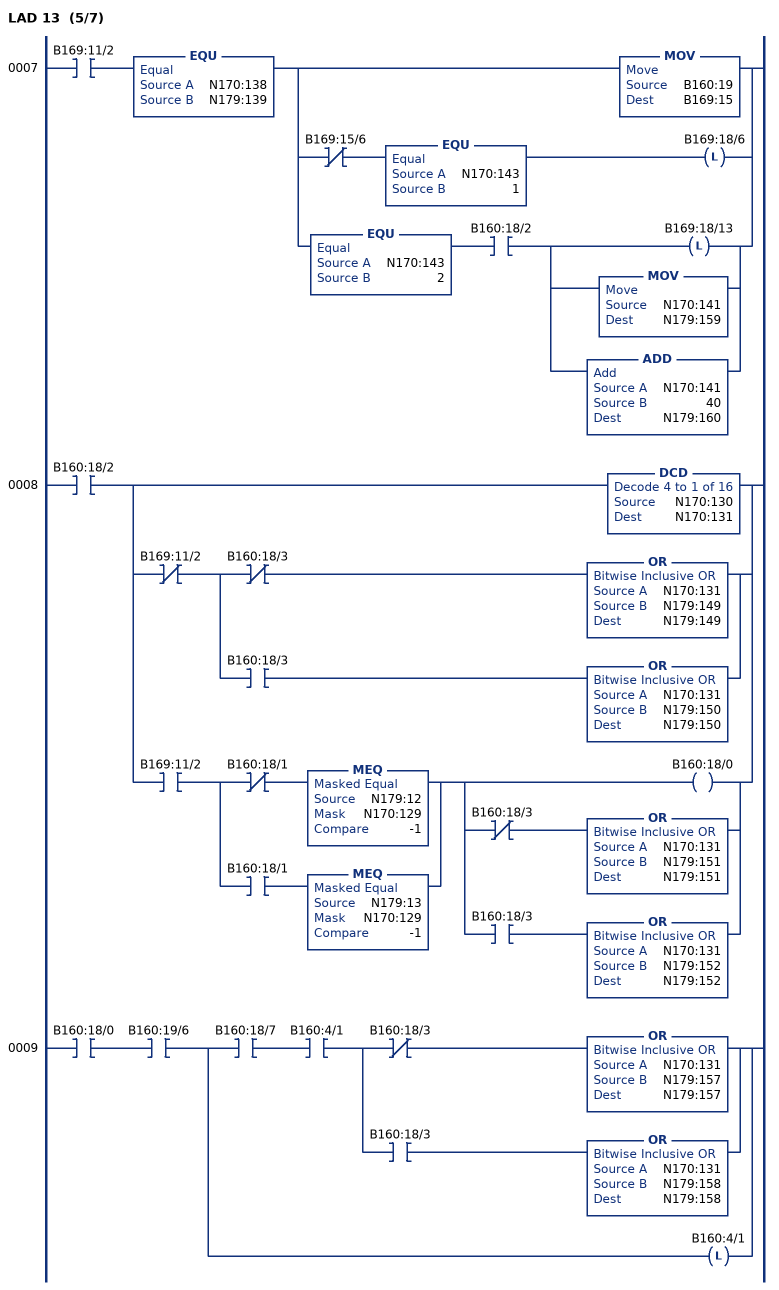
% Rung: 7 %
SOR XIC B169:11/2 EQU N170:138 N179:139 BST MOV B160:19 B169:15 NXB XIO B169:15/6 EQU N170:143 1 OTL B169:18/6 NXB EQU N170:143 2 XIC B160:18/2 BST OTL B169:18/13 NXB MOV N170:141 N179:159 NXB ADD N170:141 40 N179:160 BND BND EOR
% Rung: 8 %
SOR XIC B160:18/2 BST DCD N170:130 N170:131 NXB XIO B169:11/2 BST XIO B160:18/3 OR N170:131 N179:149 N179:149 NXB XIC B160:18/3 OR N170:131 N179:150 N179:150 BND NXB XIC B169:11/2 BST XIO B160:18/1 MEQ N179:12 N170:129 -1 NXB XIC B160:18/1 MEQ N179:13 N170:129 -1 BND BST OTE B160:18/0 NXB XIO B160:18/3 OR N170:131 N179:151 N179:151 NXB XIC B160:18/3 OR N170:131 N179:152 N179:152 BND BND EOR
% Rung: 9 %
SOR XIC B160:18/0 XIC B160:19/6 BST XIC B160:18/7 XIC B160:4/1 BST XIO B160:18/3 OR N170:131 N179:157 N179:157 NXB XIC B160:18/3 OR N170:131 N179:158 N179:158 BND NXB OTL B160:4/1 BND EOR

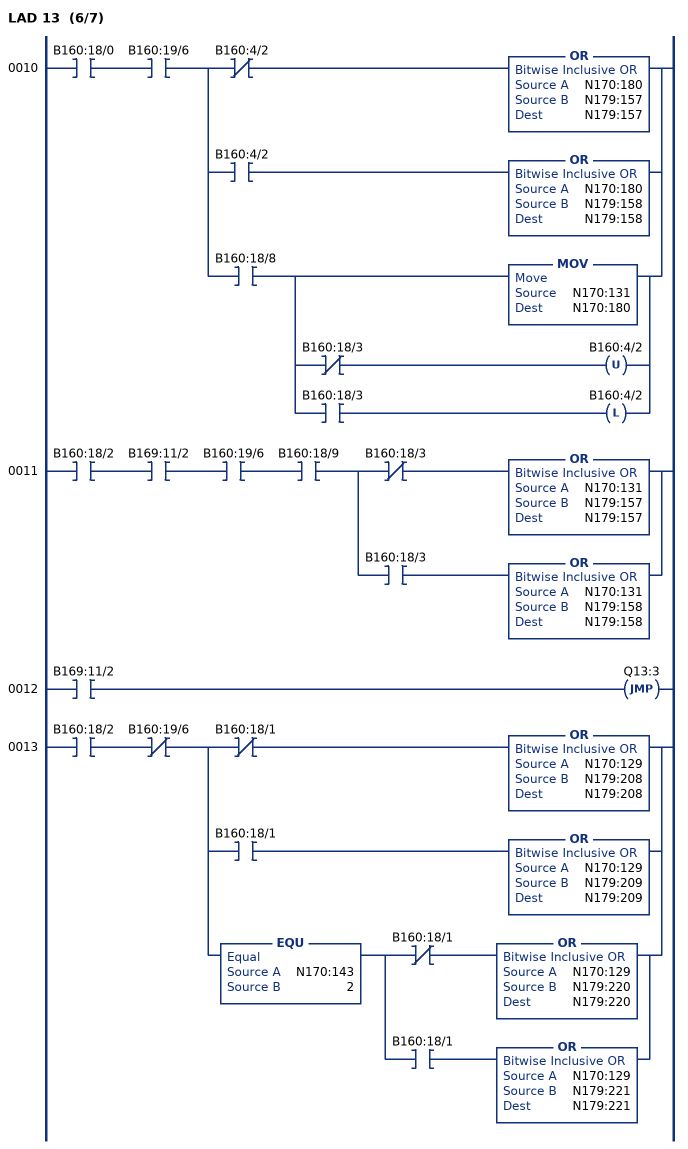
% Rung: 10 %
SOR XIC B160:18/0 XIC B160:19/6 BST BST XIO B160:4/2 OR N170:180 N179:157 N179:157 NXB XIC B160:4/2 OR N170:180 N179:158 N179:158 BND NXB XIC B160:18/8 BST MOV N170:131 N170:180 NXB XIO B160:18/3 OTU B160:4/2 NXB XIC B160:18/3 OTL B160:4/2 BND BND EOR
% Rung: 11 %
SOR XIC B160:18/2 XIC B169:11/2 XIC B160:19/6 XIC B160:18/9 BST XIO B160:18/3 OR N170:131 N179:157 N179:157 NXB XIC B160:18/3 OR N170:131 N179:158 N179:158 BND EOR
% Rung: 12 %
SOR XIC B169:11/2 JMP Q13:3 EOR
% Rung: 13 %
SOR XIC B160:18/2 XIO B160:19/6 BST BST XIO B160:18/1 OR N170:129 N179:208 N179:208 NXB XIC B160:18/1 OR N170:129 N179:209 N179:209 BND NXB EQU N170:143 2 BST XIO B160:18/1 OR N170:129 N179:220 N179:220 NXB XIC B160:18/1 OR N170:129 N179:221 N179:221 BND BND EOR

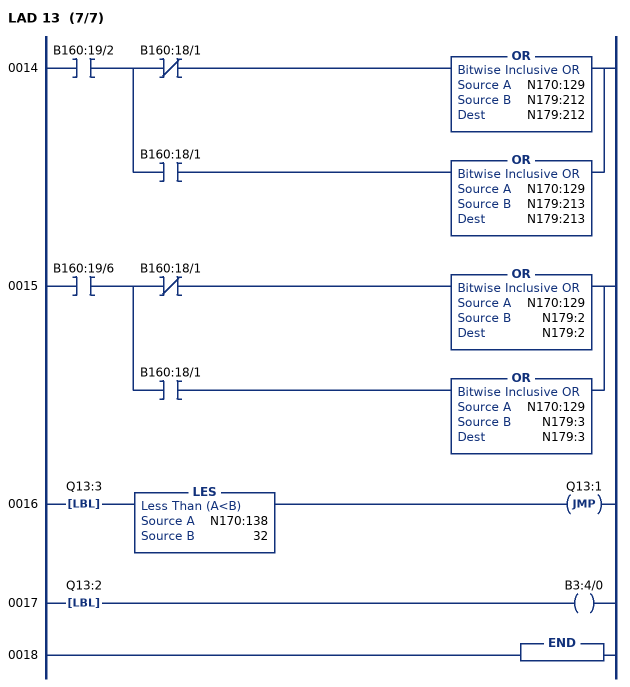
% Rung: 14 %
SOR XIC B160:19/2 BST XIO B160:18/1 OR N170:129 N179:212 N179:212 NXB XIC B160:18/1 OR N170:129 N179:213 N179:213 BND EOR
% Rung: 15 %
SOR XIC B160:19/6 BST XIO B160:18/1 OR N170:129 N179:2 N179:2 NXB XIC B160:18/1 OR N170:129 N179:3 N179:3 BND EOR
% Rung: 16 %
SOR LBL Q13:3 LES N170:138 32 JMP Q13:1 EOR
% Rung: 17 %
SOR LBL Q13:2 OTE B3:4/0 EOR
% Rung: 18 %
SOR END EOR

LADDER 15
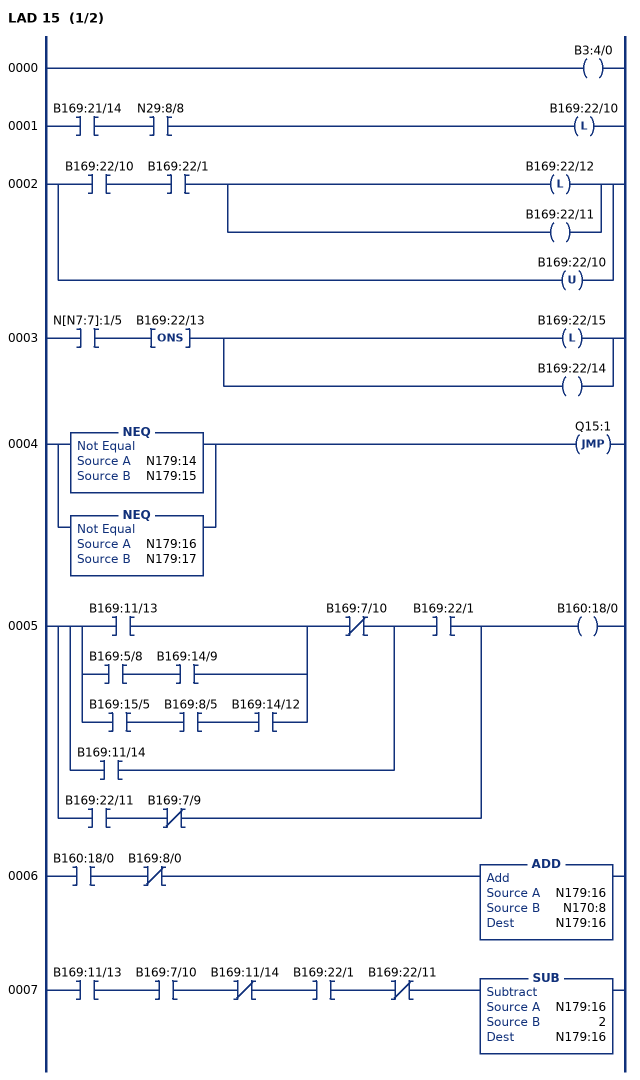
% Rung: 0 %
SOR OTE B3:4/0 EOR
% Rung: 1 %
SOR XIC B169:21/14 XIC N29:8/8 OTL B169:22/10 EOR
% Rung: 2 %
SOR BST XIC B169:22/10 XIC B169:22/1 BST OTL B169:22/12 NXB OTE B169:22/11 BND NXB OTU B169:22/10 BND EOR
% Rung: 3 %
SOR XIC N[N7:7]:1/5 OSR B169:22/13 BST OTL B169:22/15 NXB OTE B169:22/14 BND EOR
% Rung: 4 %
SOR BST NEQ N179:14 N179:15 NXB NEQ N179:16 N179:17 BND JMP Q15:1 EOR
% Rung: 5 %
SOR BST BST BST XIC B169:11/13 NXB XIC B169:5/8 XIC B169:14/9 NXB XIC B169:15/5 XIC B169:8/5 XIC B169:14/12 BND XIO B169:7/10 NXB XIC B169:11/14 BND XIC B169:22/1 NXB XIC B169:22/11 XIO B169:7/9 BND OTE B160:18/0 EOR
% Rung: 6 %
SOR XIC B160:18/0 XIO B169:8/0 ADD N179:16 N170:8 N179:16 EOR
% Rung: 7 %
SOR XIC B169:11/13 XIC B169:7/10 XIO B169:11/14 XIC B169:22/1 XIO B169:22/11 SUB N179:16 2 N179:16 EOR

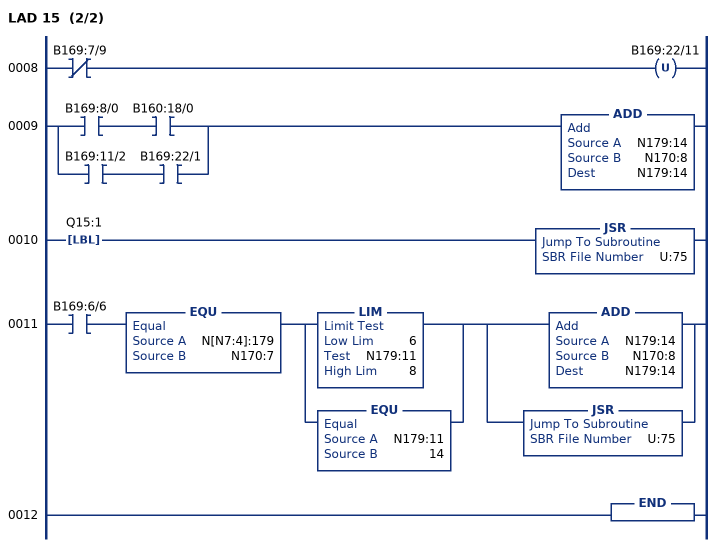
% Rung: 8 %
SOR XIO B169:7/9 OTU B169:22/11 EOR
% Rung: 9 %
SOR BST XIC B169:8/0 XIC B160:18/0 NXB XIC B169:11/2 XIC B169:22/1 BND ADD N179:14 N170:8 N179:14 EOR
% Rung: 10 %
SOR LBL Q15:1 JSR U:75 EOR
% Rung: 11 %
SOR XIC B169:6/6 EQU N[N7:4]:179 N170:7 BST LIM 6 N179:11 8 NXB EQU N179:11 14 BND BST ADD N179:14 N170:8 N179:14 NXB JSR U:75 BND EOR
% Rung: 12 %
SOR END EOR

LADDER 16
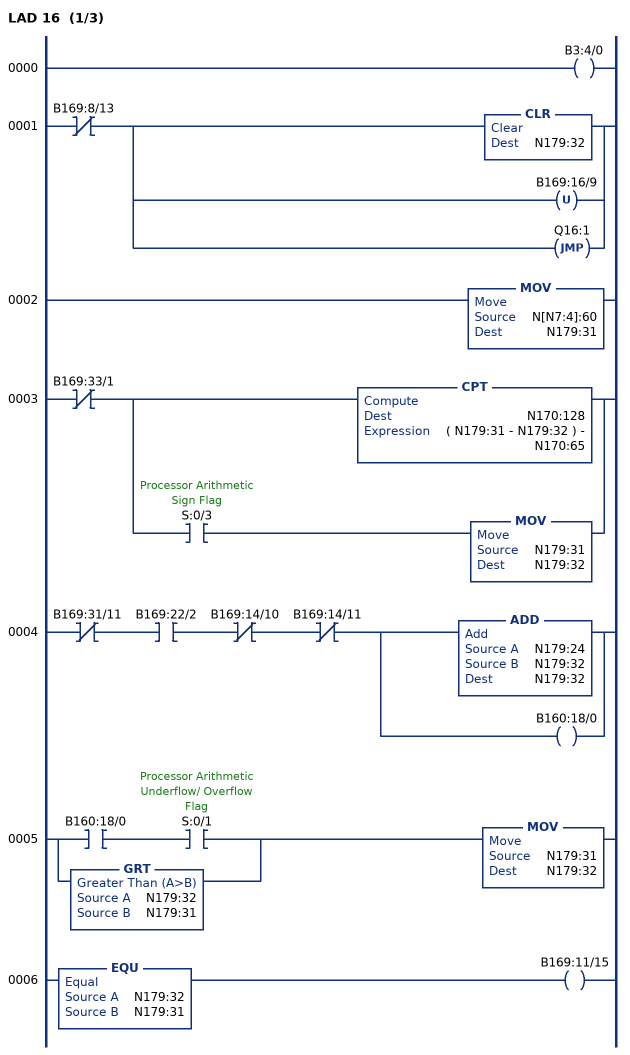
% Rung: 0 %
SOR OTE B3:4/0 EOR
% Rung: 1 %
SOR XIO B169:8/13 BST CLR N179:32 NXB OTU B169:16/9 NXB JMP Q16:1 BND EOR
% Rung: 2 %
SOR MOV N[N7:4]:60 N179:31 EOR
% Rung: 3 %
SOR XIO B169:33/1 BST CPT N170:128 " ( N179:31 - N179:32 ) - N170:65 " NXB XIC S:0/3 MOV N179:31 N179:32 BND EOR
%   S:0/3  "Processor Arithmetic Sign Flag" %
% Rung: 4 %
SOR XIO B169:31/11 XIC B169:22/2 XIO B169:14/10 XIO B169:14/11 BST ADD N179:24 N179:32 N179:32 NXB OTE B160:18/0 BND EOR
% Rung: 5 %
SOR BST XIC B160:18/0 XIC S:0/1 NXB GRT N179:32 N179:31 BND MOV N179:31 N179:32 EOR
%   S:0/1  "Processor Arithmetic Underflow/ Overflow Flag" %
% Rung: 6 %
SOR EQU N179:32 N179:31 OTE B169:11/15 EOR

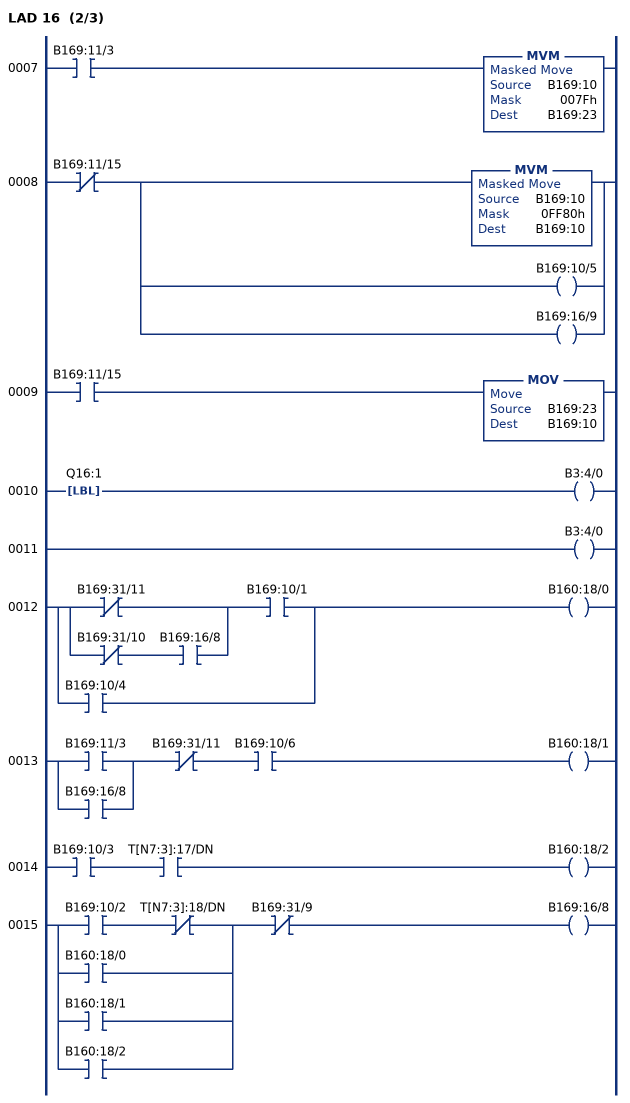
% Rung: 7 %
SOR XIC B169:11/3 MVM B169:10 007Fh B169:23 EOR
% Rung: 8 %
SOR XIO B169:11/15 BST MVM B169:10 0FF80h B169:10 NXB OTE B169:10/5 NXB OTE B169:16/9 BND EOR
% Rung: 9 %
SOR XIC B169:11/15 MOV B169:23 B169:10 EOR
% Rung: 10 %
SOR LBL Q16:1 OTE B3:4/0 EOR
% Rung: 11 %
SOR OTE B3:4/0 EOR
% Rung: 12 %
SOR BST BST XIO B169:31/11 NXB XIO B169:31/10 XIC B169:16/8 BND XIC B169:10/1 NXB XIC B169:10/4 BND OTE B160:18/0 EOR
% Rung: 13 %
SOR BST XIC B169:11/3 NXB XIC B169:16/8 BND XIO B169:31/11 XIC B169:10/6 OTE B160:18/1 EOR
% Rung: 14 %
SOR XIC B169:10/3 XIC T[N7:3]:17/DN OTE B160:18/2 EOR
% Rung: 15 %
SOR BST XIC B169:10/2 XIO T[N7:3]:18/DN NXB XIC B160:18/0 NXB XIC B160:18/1 NXB XIC B160:18/2 BND XIO B169:31/9 OTE B169:16/8 EOR

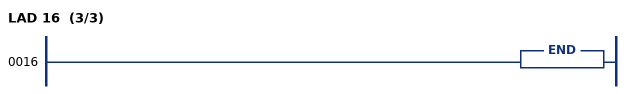
% Rung: 16 %
SOR END EOR

LADDER 17
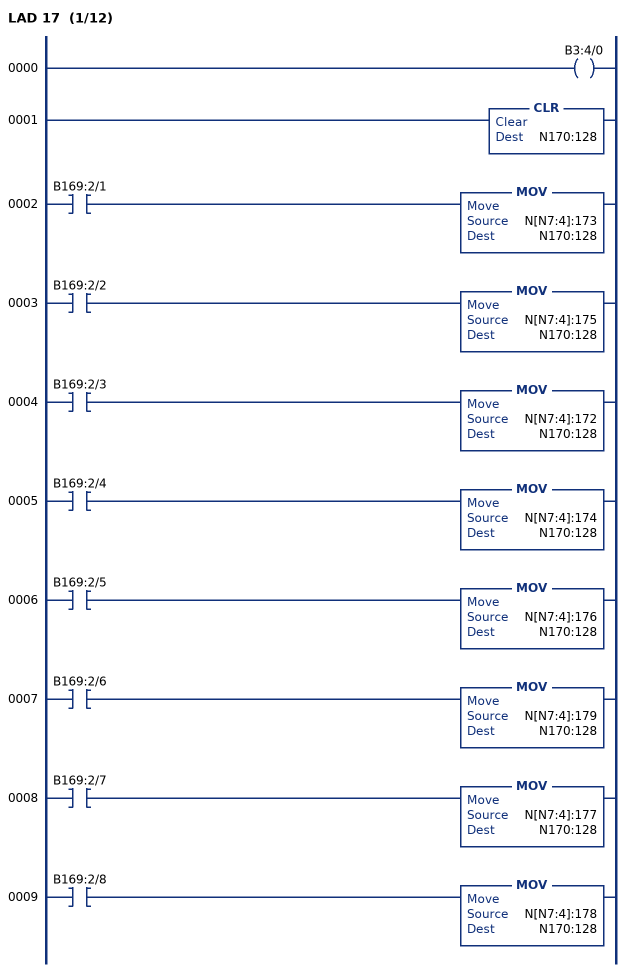
% Rung: 0 %
SOR OTE B3:4/0 EOR
% Rung: 1 %
SOR CLR N170:128 EOR
% Rung: 2 %
SOR XIC B169:2/1 MOV N[N7:4]:173 N170:128 EOR
% Rung: 3 %
SOR XIC B169:2/2 MOV N[N7:4]:175 N170:128 EOR
% Rung: 4 %
SOR XIC B169:2/3 MOV N[N7:4]:172 N170:128 EOR
% Rung: 5 %
SOR XIC B169:2/4 MOV N[N7:4]:174 N170:128 EOR
% Rung: 6 %
SOR XIC B169:2/5 MOV N[N7:4]:176 N170:128 EOR
% Rung: 7 %
SOR XIC B169:2/6 MOV N[N7:4]:179 N170:128 EOR
% Rung: 8 %
SOR XIC B169:2/7 MOV N[N7:4]:177 N170:128 EOR
% Rung: 9 %
SOR XIC B169:2/8 MOV N[N7:4]:178 N170:128 EOR

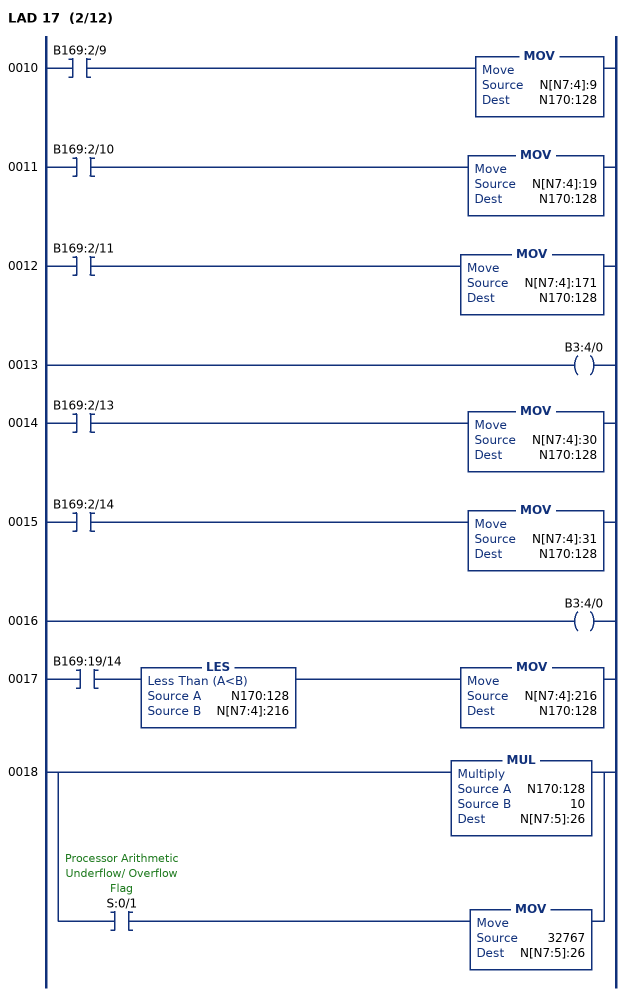
% Rung: 10 %
SOR XIC B169:2/9 MOV N[N7:4]:9 N170:128 EOR
% Rung: 11 %
SOR XIC B169:2/10 MOV N[N7:4]:19 N170:128 EOR
% Rung: 12 %
SOR XIC B169:2/11 MOV N[N7:4]:171 N170:128 EOR
% Rung: 13 %
SOR OTE B3:4/0 EOR
% Rung: 14 %
SOR XIC B169:2/13 MOV N[N7:4]:30 N170:128 EOR
% Rung: 15 %
SOR XIC B169:2/14 MOV N[N7:4]:31 N170:128 EOR
% Rung: 16 %
SOR OTE B3:4/0 EOR
% Rung: 17 %
SOR XIC B169:19/14 LES N170:128 N[N7:4]:216 MOV N[N7:4]:216 N170:128 EOR
% Rung: 18 %
SOR BST MUL N170:128 10 N[N7:5]:26 NXB XIC S:0/1 MOV 32767 N[N7:5]:26 BND EOR
%   S:0/1  "Processor Arithmetic Underflow/ Overflow Flag" %

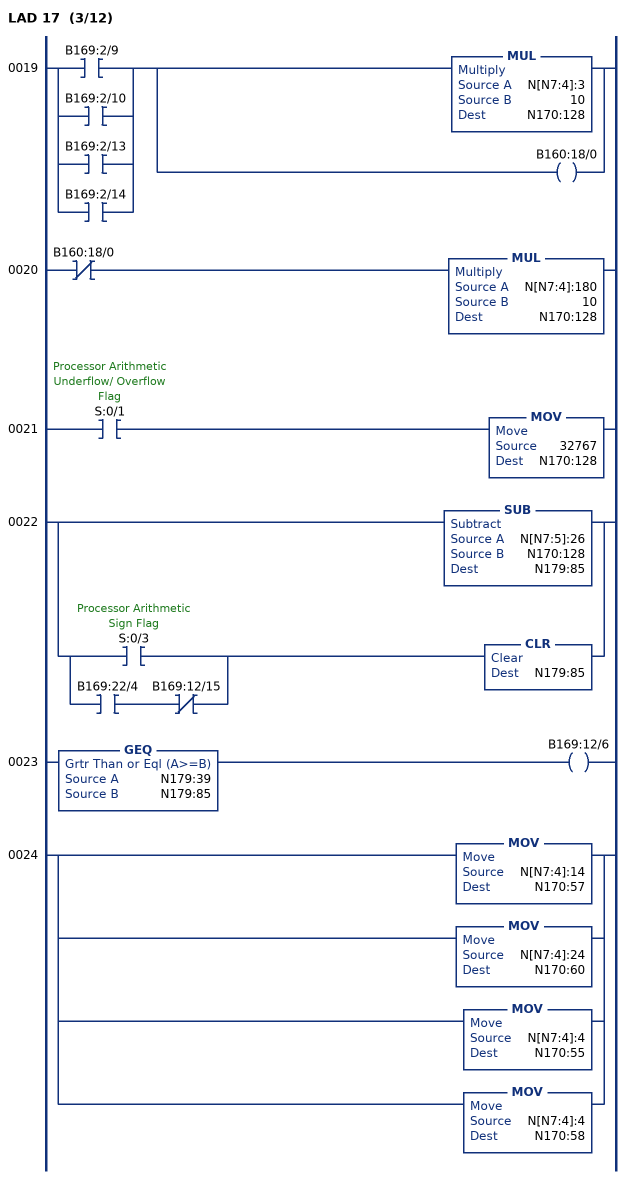
% Rung: 19 %
SOR BST XIC B169:2/9 NXB XIC B169:2/10 NXB XIC B169:2/13 NXB XIC B169:2/14 BND BST MUL N[N7:4]:3 10 N170:128 NXB OTE B160:18/0 BND EOR
% Rung: 20 %
SOR XIO B160:18/0 MUL N[N7:4]:180 10 N170:128 EOR
% Rung: 21 %
SOR XIC S:0/1 MOV 32767 N170:128 EOR
%   S:0/1  "Processor Arithmetic Underflow/ Overflow Flag" %
% Rung: 22 %
SOR BST SUB N[N7:5]:26 N170:128 N179:85 NXB BST XIC S:0/3 NXB XIC B169:22/4 XIO B169:12/15 BND CLR N179:85 BND EOR
%   S:0/3  "Processor Arithmetic Sign Flag" %
% Rung: 23 %
SOR GEQ N179:39 N179:85 OTE B169:12/6 EOR
% Rung: 24 %
SOR BST MOV N[N7:4]:14 N170:57 NXB MOV N[N7:4]:24 N170:60 NXB MOV N[N7:4]:4 N170:55 NXB MOV N[N7:4]:4 N170:58 BND EOR

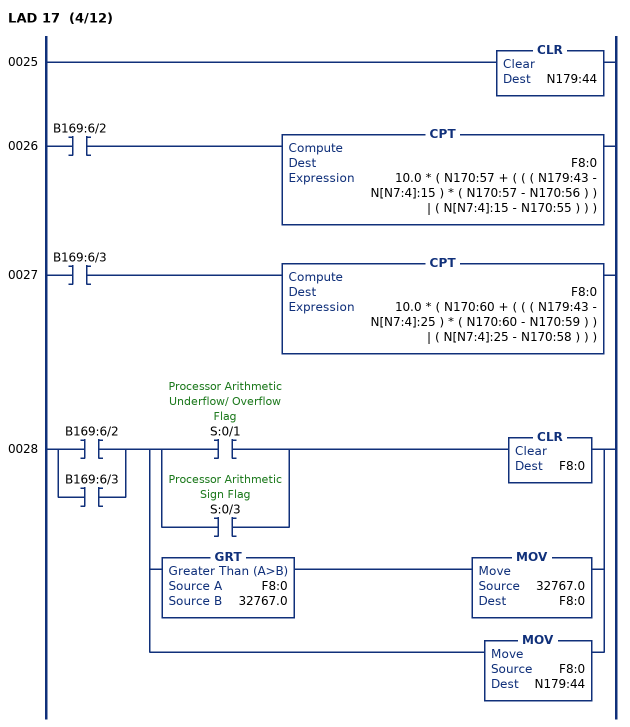
% Rung: 25 %
SOR CLR N179:44 EOR
% Rung: 26 %
SOR XIC B169:6/2 CPT F8:0 " 10.0 * ( N170:57 + ( ( ( N179:43 - N[N7:4]:15 ) * ( N170:57 - N170:56 ) ) | ( N[N7:4]:15 - N170:55 ) ) ) " EOR
% Rung: 27 %
SOR XIC B169:6/3 CPT F8:0 " 10.0 * ( N170:60 + ( ( ( N179:43 - N[N7:4]:25 ) * ( N170:60 - N170:59 ) ) | ( N[N7:4]:25 - N170:58 ) ) ) " EOR
% Rung: 28 %
SOR BST XIC B169:6/2 NXB XIC B169:6/3 BND BST BST XIC S:0/1 NXB XIC S:0/3 BND CLR F8:0 NXB GRT F8:0 32767.0 MOV 32767.0 F8:0 NXB MOV F8:0 N179:44 BND EOR
%   S:0/1  "Processor Arithmetic Underflow/ Overflow Flag" %
%   S:0/3  "Processor Arithmetic Sign Flag" %

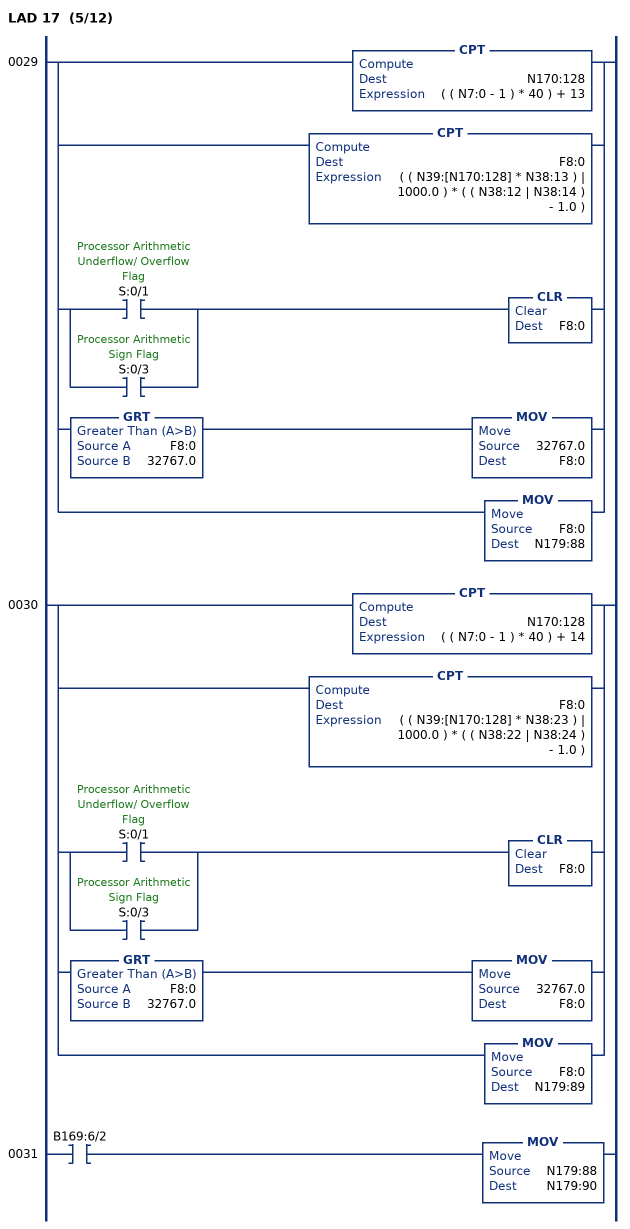
% Rung: 29 %
SOR BST CPT N170:128 " ( ( N7:0 - 1 ) * 40 ) + 13 " NXB CPT F8:0 " ( ( N39:[N170:128] * N38:13 ) | 1000.0 ) * ( ( N38:12 | N38:14 ) - 1.0 ) " NXB BST XIC S:0/1 NXB XIC S:0/3 BND CLR F8:0 NXB GRT F8:0 32767.0 MOV 32767.0 F8:0 NXB MOV F8:0 N179:88 BND EOR
%   S:0/1  "Processor Arithmetic Underflow/ Overflow Flag" %
%   S:0/3  "Processor Arithmetic Sign Flag" %
% Rung: 30 %
SOR BST CPT N170:128 " ( ( N7:0 - 1 ) * 40 ) + 14 " NXB CPT F8:0 " ( ( N39:[N170:128] * N38:23 ) | 1000.0 ) * ( ( N38:22 | N38:24 ) - 1.0 ) " NXB BST XIC S:0/1 NXB XIC S:0/3 BND CLR F8:0 NXB GRT F8:0 32767.0 MOV 32767.0 F8:0 NXB MOV F8:0 N179:89 BND EOR
%   S:0/1  "Processor Arithmetic Underflow/ Overflow Flag" %
%   S:0/3  "Processor Arithmetic Sign Flag" %
% Rung: 31 %
SOR XIC B169:6/2 MOV N179:88 N179:90 EOR

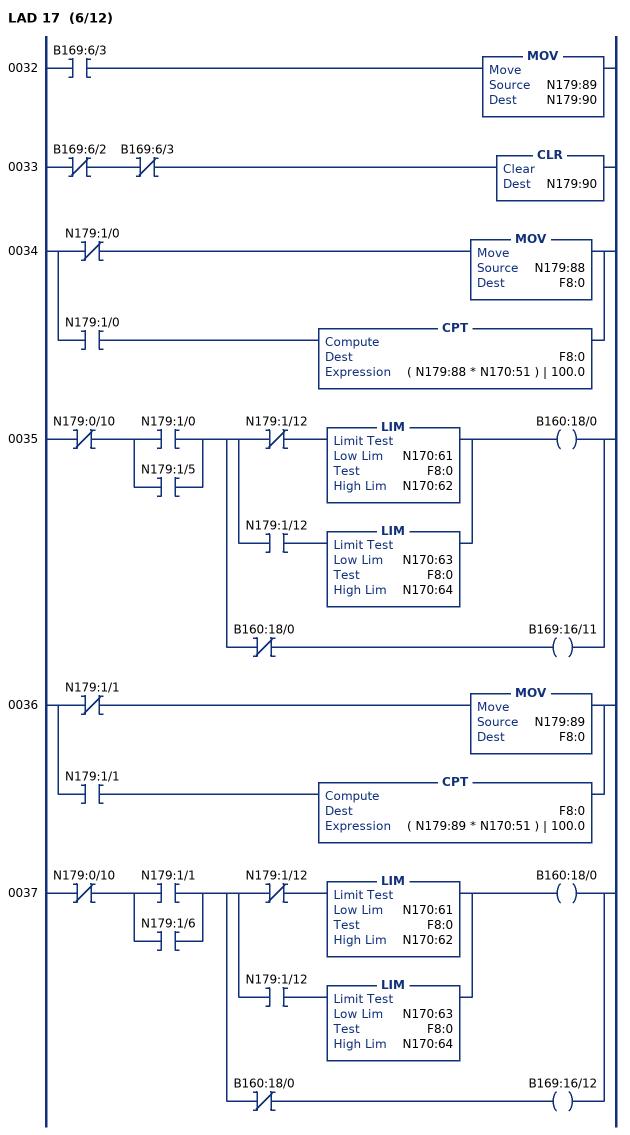
% Rung: 32 %
SOR XIC B169:6/3 MOV N179:89 N179:90 EOR
% Rung: 33 %
SOR XIO B169:6/2 XIO B169:6/3 CLR N179:90 EOR
% Rung: 34 %
SOR BST XIO N179:1/0 MOV N179:88 F8:0 NXB XIC N179:1/0 CPT F8:0 " ( N179:88 * N170:51 ) | 100.0 " BND EOR
% Rung: 35 %
SOR XIO N179:0/10 BST XIC N179:1/0 NXB XIC N179:1/5 BND BST BST XIO N179:1/12 LIM N170:61 F8:0 N170:62 NXB XIC N179:1/12 LIM N170:63 F8:0 N170:64 BND OTE B160:18/0 NXB XIO B160:18/0 OTE B169:16/11 BND EOR
% Rung: 36 %
SOR BST XIO N179:1/1 MOV N179:89 F8:0 NXB XIC N179:1/1 CPT F8:0 " ( N179:89 * N170:51 ) | 100.0 " BND EOR
% Rung: 37 %
SOR XIO N179:0/10 BST XIC N179:1/1 NXB XIC N179:1/6 BND BST BST XIO N179:1/12 LIM N170:61 F8:0 N170:62 NXB XIC N179:1/12 LIM N170:63 F8:0 N170:64 BND OTE B160:18/0 NXB XIO B160:18/0 OTE B169:16/12 BND EOR

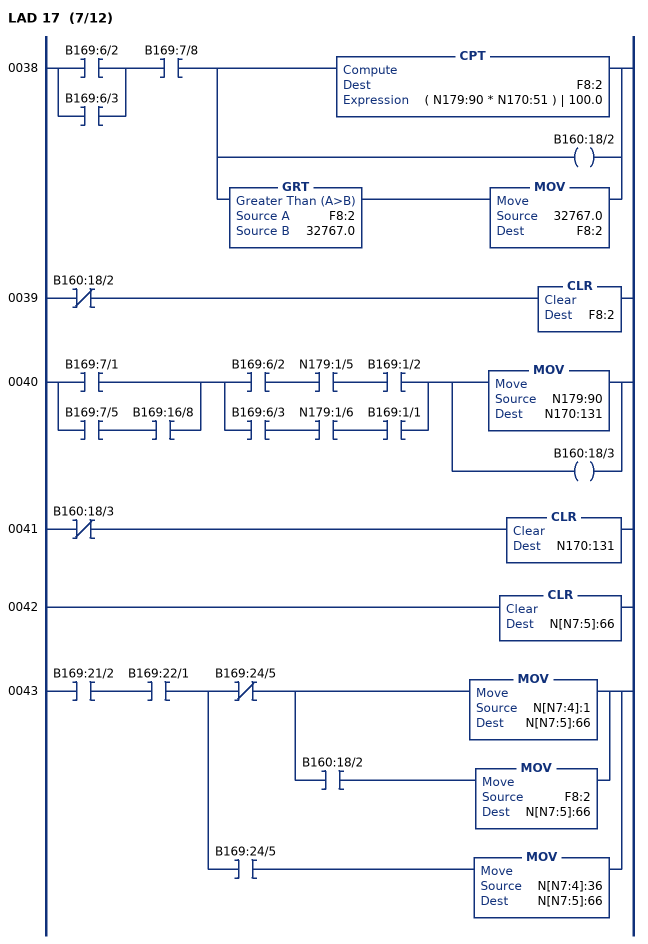
% Rung: 38 %
SOR BST XIC B169:6/2 NXB XIC B169:6/3 BND XIC B169:7/8 BST CPT F8:2 " ( N179:90 * N170:51 ) | 100.0 " NXB OTE B160:18/2 NXB GRT F8:2 32767.0 MOV 32767.0 F8:2 BND EOR
% Rung: 39 %
SOR XIO B160:18/2 CLR F8:2 EOR
% Rung: 40 %
SOR BST XIC B169:7/1 NXB XIC B169:7/5 XIC B169:16/8 BND BST XIC B169:6/2 XIC N179:1/5 XIC B169:1/2 NXB XIC B169:6/3 XIC N179:1/6 XIC B169:1/1 BND BST MOV N179:90 N170:131 NXB OTE B160:18/3 BND EOR
% Rung: 41 %
SOR XIO B160:18/3 CLR N170:131 EOR
% Rung: 42 %
SOR CLR N[N7:5]:66 EOR
% Rung: 43 %
SOR XIC B169:21/2 XIC B169:22/1 BST XIO B169:24/5 BST MOV N[N7:4]:1 N[N7:5]:66 NXB XIC B160:18/2 MOV F8:2 N[N7:5]:66 BND NXB XIC B169:24/5 MOV N[N7:4]:36 N[N7:5]:66 BND EOR

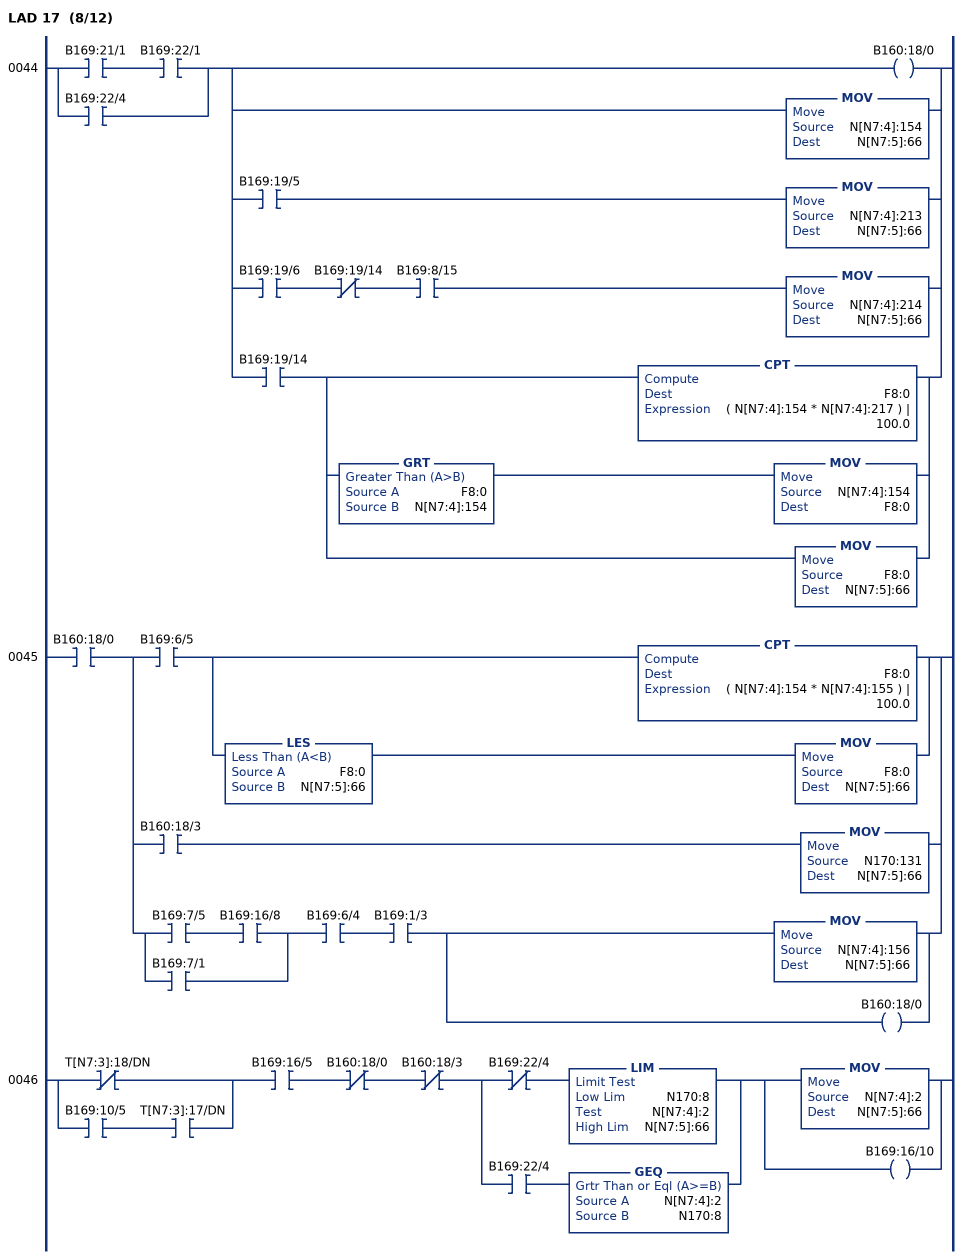
% Rung: 44 %
SOR BST XIC B169:21/1 XIC B169:22/1 NXB XIC B169:22/4 BND BST BST BST OTE B160:18/0 NXB MOV N[N7:4]:154 N[N7:5]:66 BND NXB BST XIC B169:19/5 MOV N[N7:4]:213 N[N7:5]:66 NXB XIC B169:19/6 XIO B169:19/14 XIC B169:8/15 MOV N[N7:4]:214 N[N7:5]:66 BND BND NXB XIC B169:19/14 BST CPT F8:0 " ( N[N7:4]:154 * N[N7:4]:217 ) | 100.0 " NXB GRT F8:0 N[N7:4]:154 MOV N[N7:4]:154 F8:0 NXB MOV F8:0 N[N7:5]:66 BND BND EOR
% Rung: 45 %
SOR XIC B160:18/0 BST BST XIC B169:6/5 BST CPT F8:0 " ( N[N7:4]:154 * N[N7:4]:155 ) | 100.0 " NXB LES F8:0 N[N7:5]:66 MOV F8:0 N[N7:5]:66 BND NXB XIC B160:18/3 MOV N170:131 N[N7:5]:66 BND NXB BST XIC B169:7/5 XIC B169:16/8 NXB XIC B169:7/1 BND XIC B169:6/4 XIC B169:1/3 BST MOV N[N7:4]:156 N[N7:5]:66 NXB OTE B160:18/0 BND BND EOR
% Rung: 46 %
SOR BST XIO T[N7:3]:18/DN NXB XIC B169:10/5 XIC T[N7:3]:17/DN BND XIC B169:16/5 XIO B160:18/0 XIO B160:18/3 BST XIO B169:22/4 LIM N170:8 N[N7:4]:2 N[N7:5]:66 NXB XIC B169:22/4 GEQ N[N7:4]:2 N170:8 BND BST MOV N[N7:4]:2 N[N7:5]:66 NXB OTE B169:16/10 BND EOR

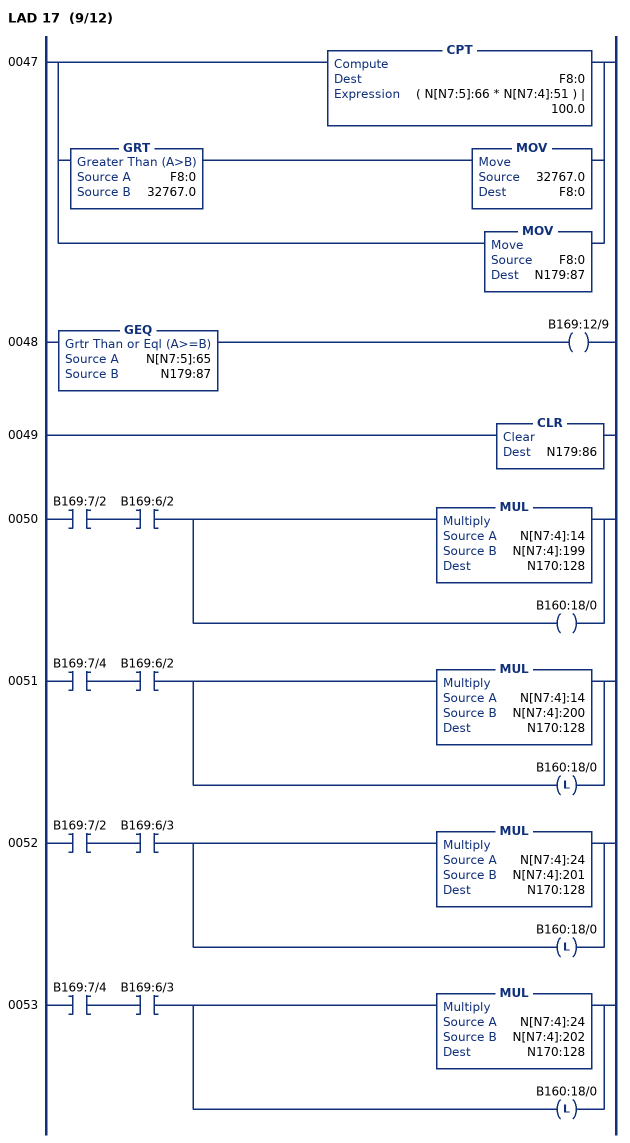
% Rung: 47 %
SOR BST CPT F8:0 " ( N[N7:5]:66 * N[N7:4]:51 ) | 100.0 " NXB GRT F8:0 32767.0 MOV 32767.0 F8:0 NXB MOV F8:0 N179:87 BND EOR
% Rung: 48 %
SOR GEQ N[N7:5]:65 N179:87 OTE B169:12/9 EOR
% Rung: 49 %
SOR CLR N179:86 EOR
% Rung: 50 %
SOR XIC B169:7/2 XIC B169:6/2 BST MUL N[N7:4]:14 N[N7:4]:199 N170:128 NXB OTE B160:18/0 BND EOR
% Rung: 51 %
SOR XIC B169:7/4 XIC B169:6/2 BST MUL N[N7:4]:14 N[N7:4]:200 N170:128 NXB OTL B160:18/0 BND EOR
% Rung: 52 %
SOR XIC B169:7/2 XIC B169:6/3 BST MUL N[N7:4]:24 N[N7:4]:201 N170:128 NXB OTL B160:18/0 BND EOR
% Rung: 53 %
SOR XIC B169:7/4 XIC B169:6/3 BST MUL N[N7:4]:24 N[N7:4]:202 N170:128 NXB OTL B160:18/0 BND EOR

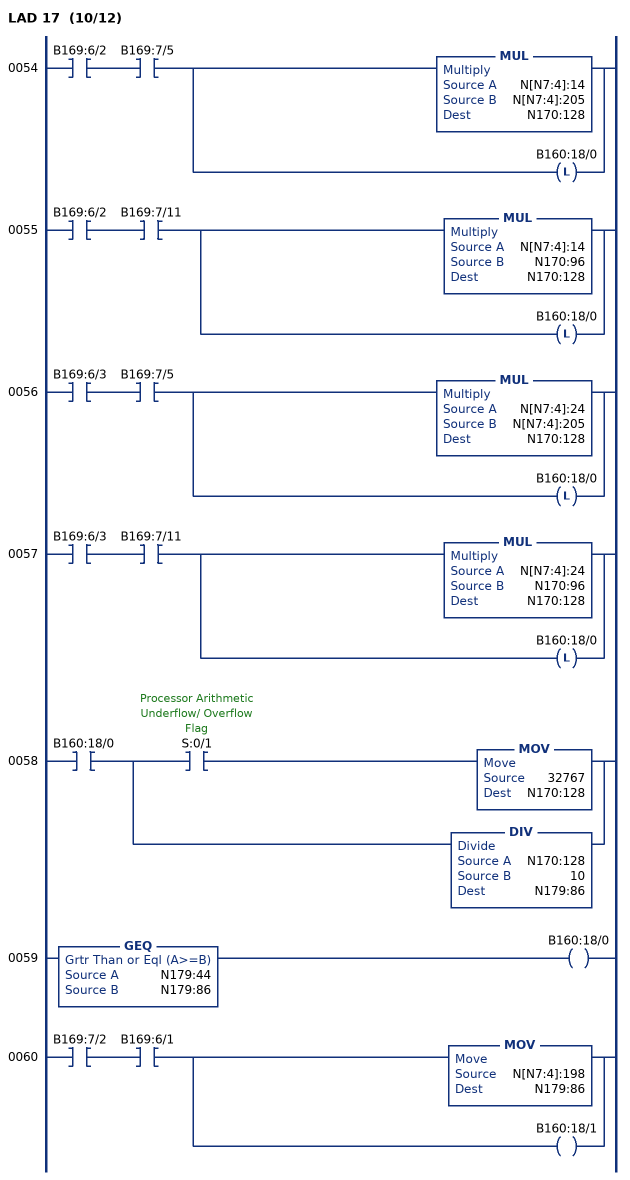
% Rung: 54 %
SOR XIC B169:6/2 XIC B169:7/5 BST MUL N[N7:4]:14 N[N7:4]:205 N170:128 NXB OTL B160:18/0 BND EOR
% Rung: 55 %
SOR XIC B169:6/2 XIC B169:7/11 BST MUL N[N7:4]:14 N170:96 N170:128 NXB OTL B160:18/0 BND EOR
% Rung: 56 %
SOR XIC B169:6/3 XIC B169:7/5 BST MUL N[N7:4]:24 N[N7:4]:205 N170:128 NXB OTL B160:18/0 BND EOR
% Rung: 57 %
SOR XIC B169:6/3 XIC B169:7/11 BST MUL N[N7:4]:24 N170:96 N170:128 NXB OTL B160:18/0 BND EOR
% Rung: 58 %
SOR XIC B160:18/0 BST XIC S:0/1 MOV 32767 N170:128 NXB DIV N170:128 10 N179:86 BND EOR
%   S:0/1  "Processor Arithmetic Underflow/ Overflow Flag" %
% Rung: 59 %
SOR GEQ N179:44 N179:86 OTE B160:18/0 EOR
% Rung: 60 %
SOR XIC B169:7/2 XIC B169:6/1 BST MOV N[N7:4]:198 N179:86 NXB OTE B160:18/1 BND EOR

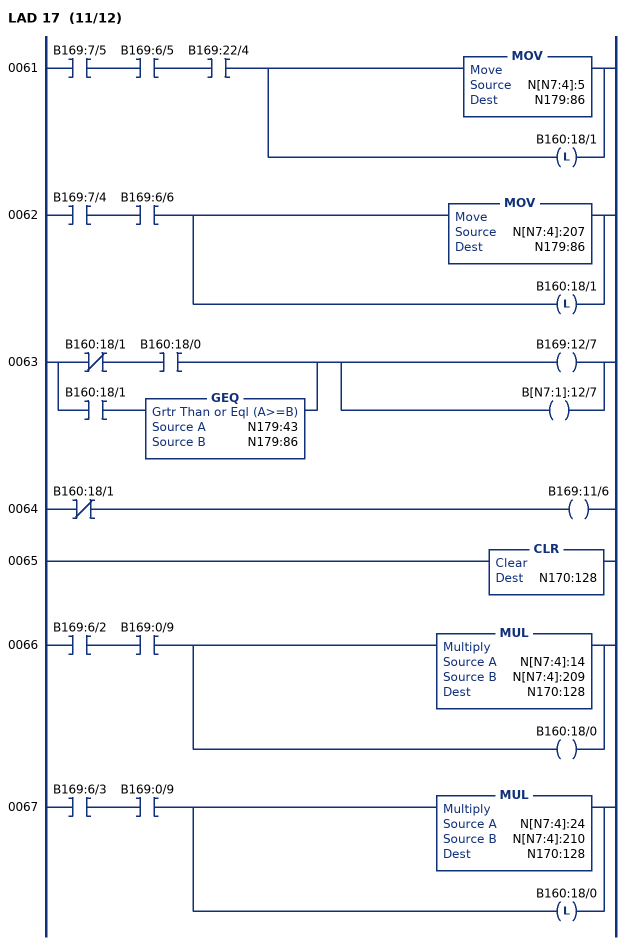
% Rung: 61 %
SOR XIC B169:7/5 XIC B169:6/5 XIC B169:22/4 BST MOV N[N7:4]:5 N179:86 NXB OTL B160:18/1 BND EOR
% Rung: 62 %
SOR XIC B169:7/4 XIC B169:6/6 BST MOV N[N7:4]:207 N179:86 NXB OTL B160:18/1 BND EOR
% Rung: 63 %
SOR BST XIO B160:18/1 XIC B160:18/0 NXB XIC B160:18/1 GEQ N179:43 N179:86 BND BST OTE B169:12/7 NXB OTE B[N7:1]:12/7 BND EOR
% Rung: 64 %
SOR XIO B160:18/1 OTE B169:11/6 EOR
% Rung: 65 %
SOR CLR N170:128 EOR
% Rung: 66 %
SOR XIC B169:6/2 XIC B169:0/9 BST MUL N[N7:4]:14 N[N7:4]:209 N170:128 NXB OTE B160:18/0 BND EOR
% Rung: 67 %
SOR XIC B169:6/3 XIC B169:0/9 BST MUL N[N7:4]:24 N[N7:4]:210 N170:128 NXB OTL B160:18/0 BND EOR

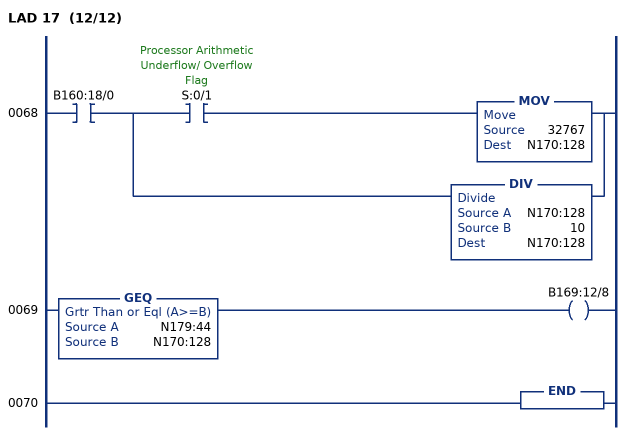
% Rung: 68 %
SOR XIC B160:18/0 BST XIC S:0/1 MOV 32767 N170:128 NXB DIV N170:128 10 N170:128 BND EOR
%   S:0/1  "Processor Arithmetic Underflow/ Overflow Flag" %
% Rung: 69 %
SOR GEQ N179:44 N170:128 OTE B169:12/8 EOR
% Rung: 70 %
SOR END EOR

LADDER 18
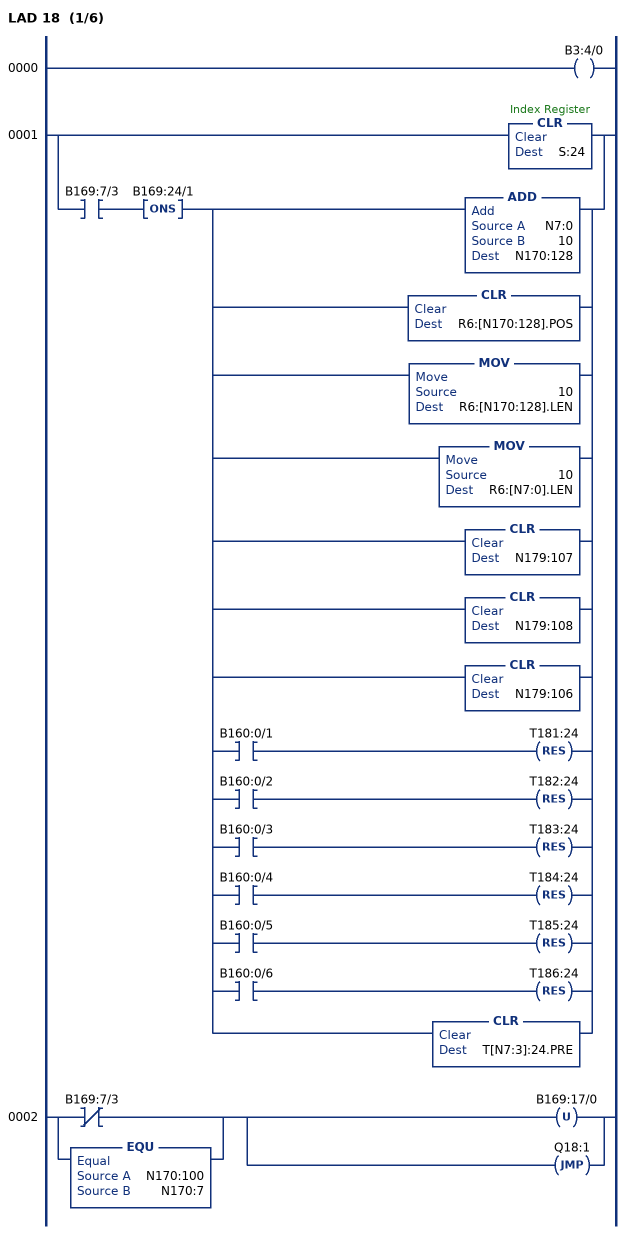
% Rung: 0 %
SOR OTE B3:4/0 EOR
% Rung: 1 %
SOR BST CLR S:24 NXB XIC B169:7/3 OSR B169:24/1 BST ADD N7:0 10 N170:128 NXB CLR R6:[N170:128].POS NXB MOV 10 R6:[N170:128].LEN NXB MOV 10 R6:[N7:0].LEN NXB CLR N179:107 NXB CLR N179:108 NXB CLR N179:106 NXB XIC B160:0/1 RES T181:24 NXB XIC B160:0/2 RES T182:24 NXB XIC B160:0/3 RES T183:24 NXB XIC B160:0/4 RES T184:24 NXB XIC B160:0/5 RES T185:24 NXB XIC B160:0/6 RES T186:24 NXB CLR T[N7:3]:24.PRE BND BND EOR
%   S:24  "Index Register" %
% Rung: 2 %
SOR BST XIO B169:7/3 NXB EQU N170:100 N170:7 BND BST OTU B169:17/0 NXB JMP Q18:1 BND EOR

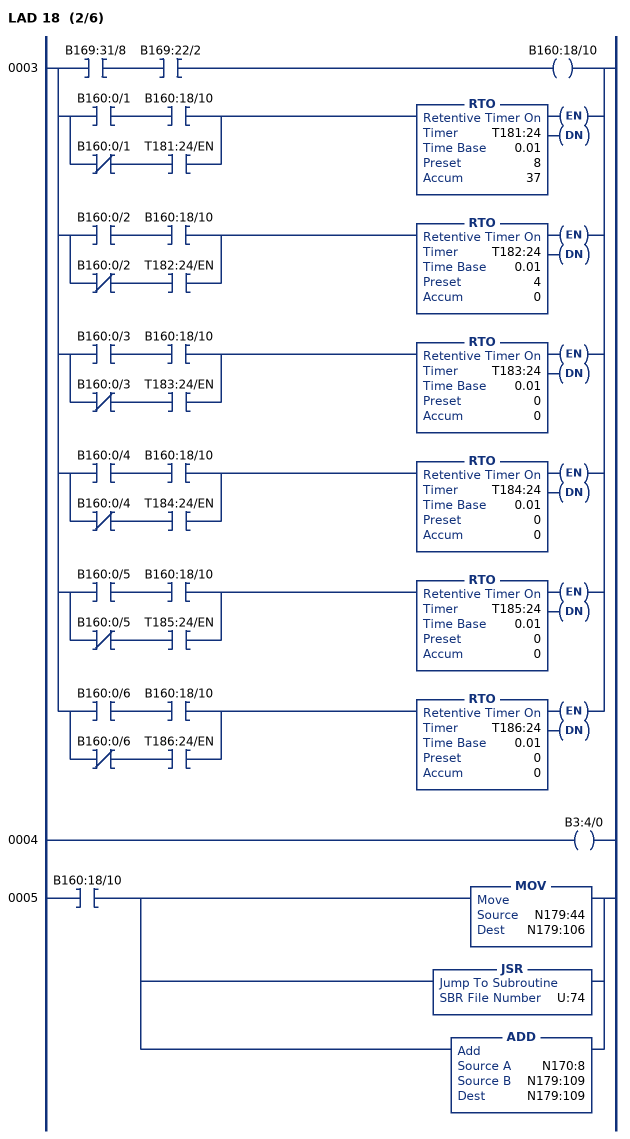
% Rung: 3 %
SOR BST XIC B169:31/8 XIC B169:22/2 OTE B160:18/10 NXB BST XIC B160:0/1 XIC B160:18/10 NXB XIO B160:0/1 XIC T181:24/EN BND RTO T181:24 0.01 8 37 NXB BST XIC B160:0/2 XIC B160:18/10 NXB XIO B160:0/2 XIC T182:24/EN BND RTO T182:24 0.01 4 0 NXB BST XIC B160:0/3 XIC B160:18/10 NXB XIO B160:0/3 XIC T183:24/EN BND RTO T183:24 0.01 0 0 NXB BST XIC B160:0/4 XIC B160:18/10 NXB XIO B160:0/4 XIC T184:24/EN BND RTO T184:24 0.01 0 0 NXB BST XIC B160:0/5 XIC B160:18/10 NXB XIO B160:0/5 XIC T185:24/EN BND RTO T185:24 0.01 0 0 NXB BST XIC B160:0/6 XIC B160:18/10 NXB XIO B160:0/6 XIC T186:24/EN BND RTO T186:24 0.01 0 0 BND EOR
% Rung: 4 %
SOR OTE B3:4/0 EOR
% Rung: 5 %
SOR XIC B160:18/10 BST MOV N179:44 N179:106 NXB JSR U:74 NXB ADD N170:8 N179:109 N179:109 BND EOR

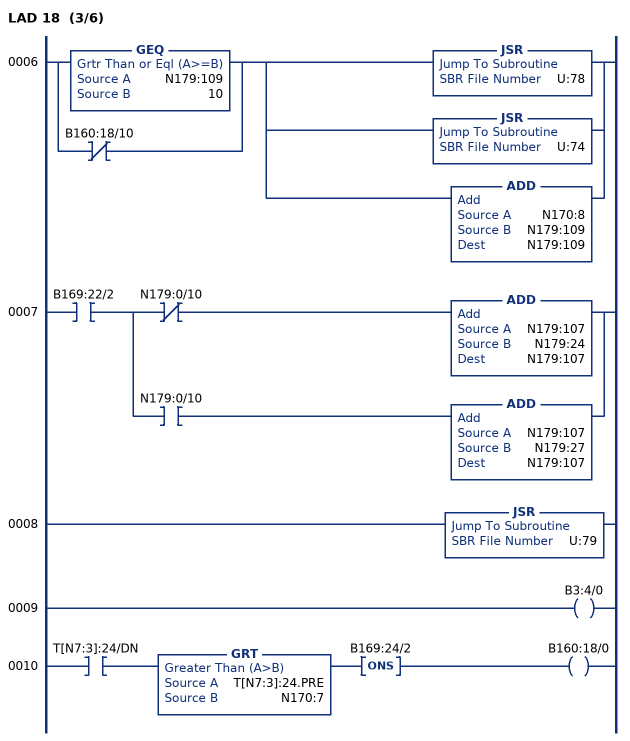
% Rung: 6 %
SOR BST GEQ N179:109 10 NXB XIO B160:18/10 BND BST JSR U:78 NXB JSR U:74 NXB ADD N170:8 N179:109 N179:109 BND EOR
% Rung: 7 %
SOR XIC B169:22/2 BST XIO N179:0/10 ADD N179:107 N179:24 N179:107 NXB XIC N179:0/10 ADD N179:107 N179:27 N179:107 BND EOR
% Rung: 8 %
SOR JSR U:79 EOR
% Rung: 9 %
SOR OTE B3:4/0 EOR
% Rung: 10 %
SOR XIC T[N7:3]:24/DN GRT T[N7:3]:24.PRE N170:7 OSR B169:24/2 OTE B160:18/0 EOR

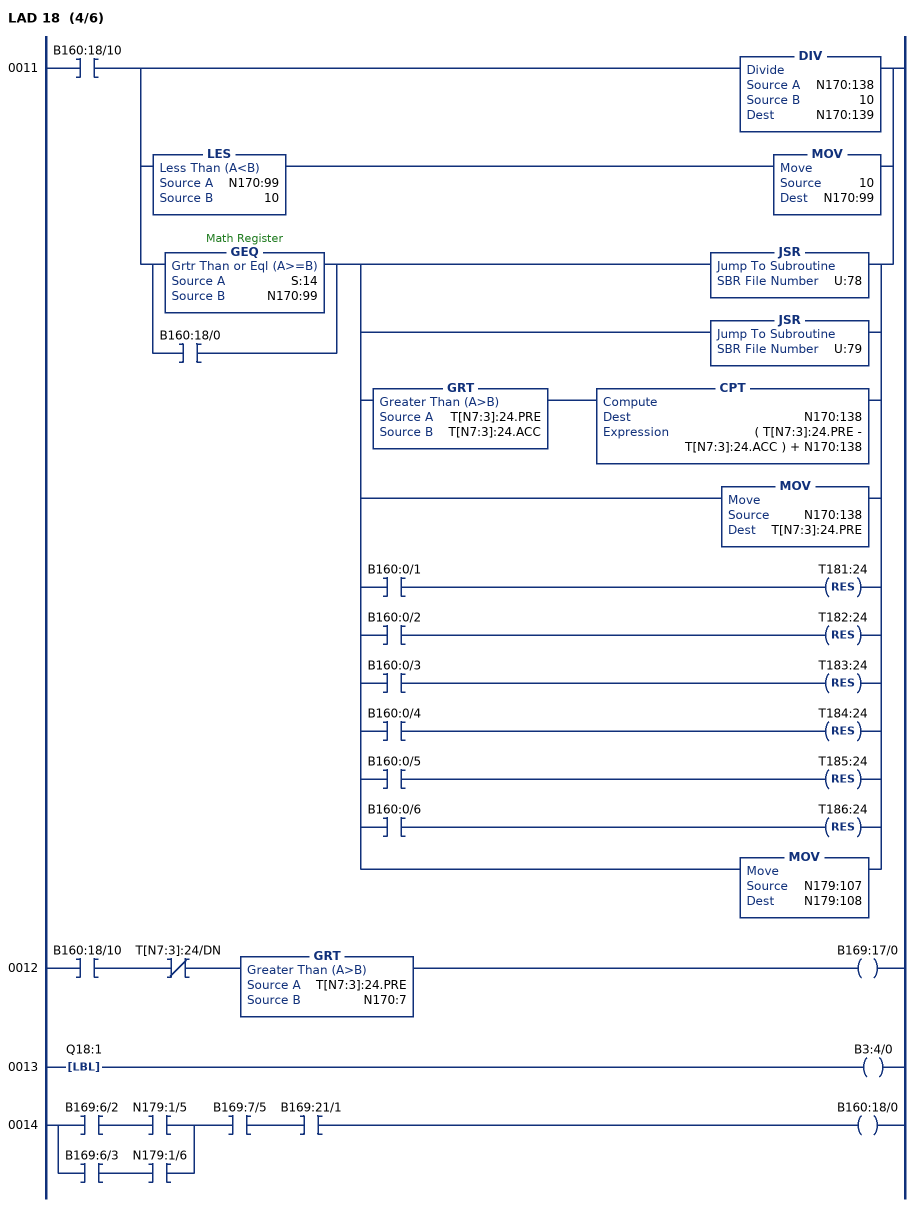
% Rung: 11 %
SOR XIC B160:18/10 BST DIV N170:138 10 N170:139 NXB LES N170:99 10 MOV 10 N170:99 NXB BST GEQ S:14 N170:99 NXB XIC B160:18/0 BND BST JSR U:78 NXB JSR U:79 NXB GRT T[N7:3]:24.PRE T[N7:3]:24.ACC CPT N170:138 " ( T[N7:3]:24.PRE - T[N7:3]:24.ACC ) + N170:138 " NXB MOV N170:138 T[N7:3]:24.PRE NXB BST XIC B160:0/1 RES T181:24 NXB XIC B160:0/2 RES T182:24 NXB XIC B160:0/3 RES T183:24 NXB XIC B160:0/4 RES T184:24 NXB XIC B160:0/5 RES T185:24 NXB XIC B160:0/6 RES T186:24 BND NXB MOV N179:107 N179:108 BND BND EOR
%   S:14  "Math Register" %
% Rung: 12 %
SOR XIC B160:18/10 XIO T[N7:3]:24/DN GRT T[N7:3]:24.PRE N170:7 OTE B169:17/0 EOR
% Rung: 13 %
SOR LBL Q18:1 OTE B3:4/0 EOR
% Rung: 14 %
SOR BST XIC B169:6/2 XIC N179:1/5 NXB XIC B169:6/3 XIC N179:1/6 BND XIC B169:7/5 XIC B169:21/1 OTE B160:18/0 EOR

